{attribute 'qualified_only'}
{attribute 'pack_mode' := '1'}
VAR_GLOBAL
			stAdsInput  AT%I* : ST_EMAdsInput;
			stAdsOutput AT%Q* : ST_EMAdsOutput;
END_VAR

(* stored: Version 1.1.0.1, ProductVersion 3.1.4024.15
   GVL EMSensor: Id {b9ae20b9-6507-47f1-9888-03b47bcef472} *)
